ABB RobotStudio station: MGietka gripper.rspag

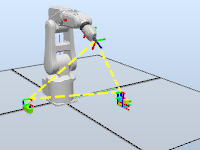
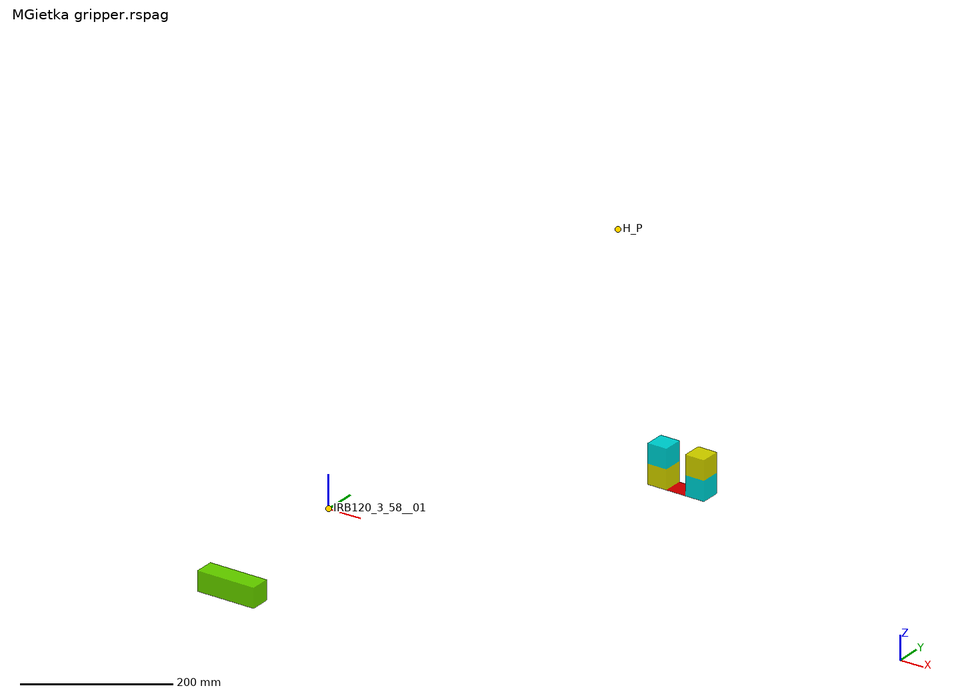
[picture v1: parts stored in the station drawn from their meshes, with robot base, taught points and paths (robot models come from the ABB library and are not in the file)]
--- station ---
Station PZPL zaliczenie 2 (saved by RobotStudio 21.4.9700.0)
Controller Controller1
  mechanical unit ROB_1: IRB120_3_58__01, 6 joints, base frame (0, 0, 0) mm
Layout (positions relative to the parent item):
  - IRB120_3_58__01 [mechanism, from Robots\IRB120_3_58_G_01.rslib] at (0, 0, 0) mm; joint values [0, 0, 0, 0, 0.5236, 0] (rad or m)
  - Smart_Gripper_Servo_Fingers [mechanism, from Tools\ABB_Smart_Gripper_Servo_Fingers.rslib] at (364.35, 0, 594) mm, rotated rx 180 ry 60 rz 180 deg; joint values [0.025] (rad or m)
  - Kosc_1 [part], size 30 x 30 x 30 mm
  - Kosc_2 [part], size 30 x 30 x 30 mm
  - Kosc_4 [part], size 30 x 30 x 30 mm
  - Kosc_3 [part], size 30 x 30 x 30 mm
  - podstawa [part], size 90 x 30 x 30 mm
  - PoseMover [smart component, from Components\PoseMover.rslib]
      properties: Mechanism=Smart_Gripper_Servo_Fingers; Pose=2; Duration=1
  - PoseMover_2 [smart component, from Components\PoseMover.rslib]
      properties: Mechanism=Smart_Gripper_Servo_Fingers; Pose=1; Duration=1
  - CollisionSensor [smart component, from Components\CollisionSensor.rslib]
      properties: Object1=Smart_Gripper_Servo_Fingers; Object2=Kosc_2; NearMiss=0; Part1=(none); Part2=(none); CollisionType=0
  - Attacher [smart component, from Components\Attacher.rslib]
      properties: Parent=Smart_Gripper_Servo_Fingers; Flange=0; Child=Kosc_2; Mount=false; Offset=[0 0 0]; Orientation=[0 0 0]
  - Detacher [smart component, from Components\Detacher.rslib]
      properties: Child=Kosc_2; KeepPosition=true
  - ClosestObject [smart component, from Components\ClosestObject.rslib]
      properties: ReferenceObject=Smart_Gripper_Servo_Fingers; ReferencePoint=[0 0 0]; RootObject=(none); ClosestObject=(none); ClosestPart=(none); Distance=0
  - plaszczyzna [part], size 90 x 30 x 0 mm
Attachment: Smart_Gripper_Servo_Fingers is attached to IRB120_3_58__01 / Link6
Attachment: Kosc1 is attached to Kosc_1
Attachment: Kosc_2 is attached to Kosc_2
Attachment: Kosc_3 is attached to Kosc_3
Attachment: Kosc_4 is attached to Kosc_4
Attachment: Podstawa is attached to podstawa
Attachment: Ramie is attached to IRB120_3_58__01 / Base
Station signals: DI start_s
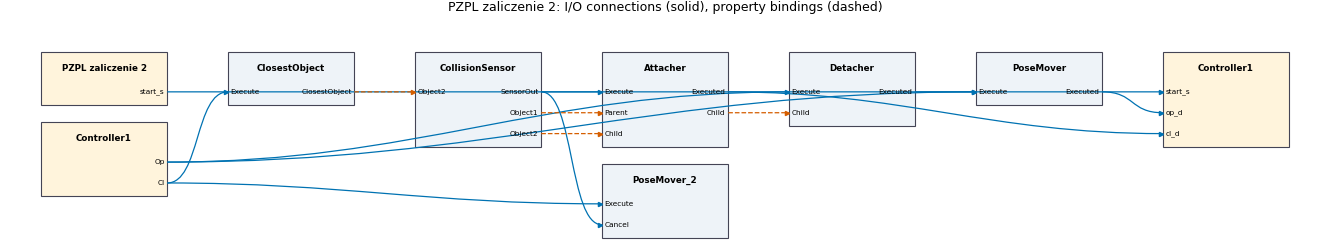
Station logic (signal -> signal, property => property):
  PZPL zaliczenie 2.start_s -> Controller1.start_s
  Controller1.Op -> PoseMover.Execute
  Controller1.Cl -> PoseMover_2.Execute
  CollisionSensor.SensorOut -> Attacher.Execute
  PoseMover.Executed -> Controller1.op_d
  CollisionSensor.SensorOut -> PoseMover_2.Cancel
  Controller1.Op -> Detacher.Execute
  Detacher.Executed -> PoseMover.Execute
  Attacher.Executed -> Controller1.cl_d
  Controller1.Cl -> ClosestObject.Execute
  CollisionSensor.Object1 => Attacher.Parent
  CollisionSensor.Object2 => Attacher.Child
  Attacher.Child => Detacher.Child
  ClosestObject.ClosestObject => CollisionSensor.Object2

--- Backups/Controller1/RAPID/TASK1/PROGMOD/CalibData.mod ---
MODULE CalibData
    PERS tooldata Servo:=[TRUE,[[0,0,114.2],[1,0,0,0]],[0.215,[8.7,12.3,49.2],[1,0,0,0],0.00021,0.00024,0.00009]];
    TASK PERS wobjdata Kosc1:=[FALSE,TRUE,"",[[300,300,0],[1,0,0,0]],[[0,0,0],[1,0,0,0]]];
    TASK PERS wobjdata Kosc_2:=[FALSE,TRUE,"",[[300,300,30],[1,0,0,0]],[[0,0,0],[1,0,0,0]]];
    TASK PERS wobjdata Kosc_3:=[FALSE,TRUE,"",[[360,300,0],[1,0,0,0]],[[0,0,0],[1,0,0,0]]];
    TASK PERS wobjdata Kosc_4:=[FALSE,TRUE,"",[[360,300,30],[1,0,0,0]],[[0,0,0],[1,0,0,0]]];
    TASK PERS wobjdata Podstawa:=[FALSE,TRUE,"",[[0,-300,0],[1,0,0,0]],[[0,0,0],[1,0,0,0]]];
    TASK PERS wobjdata Ramie:=[FALSE,TRUE,"",[[0,0,0],[1,0,0,0]],[[0,0,0],[1,0,0,0]]];
ENDMODULE

--- Backups/Controller1/RAPID/TASK1/PROGMOD/Module1.mod ---
MODULE Module1
    CONST robtarget H_P:=[[463.253930185,0,536.9],[0.5,0,0.866025404,0],[0,0,0,0],[9E+09,9E+09,9E+09,9E+09,9E+09,9E+09]];
    VAR robtarget Nad_kosc:=[[15,15,160],[0,1,0,0],[0,0,-2,0],[9E+09,9E+09,9E+09,9E+09,9E+09,9E+09]];
    VAR robtarget Kosc:=[[15,15,30],[0,1,0,0],[0,0,-2,0],[9E+09,9E+09,9E+09,9E+09,9E+09,9E+09]];
    VAR robtarget nad_cel:=[[75,15,160],[0,1,0,0],[-1,0,1,0],[9E+09,9E+09,9E+09,9E+09,9E+09,9E+09]];
    VAR robtarget cel:=[[75,15,60],[0,1,0,0],[-1,0,1,0],[9E+09,9E+09,9E+09,9E+09,9E+09,9E+09]];
    VAR num ilosc := 3;
!***********************************************************
    !
    ! Module:  Module1
    !
    ! Description:
    !   <Insert description here>
    !
    ! Author: Mati
    !
    ! Version: 1.0
    !
    !***********************************************************


    !***********************************************************
    !
    ! Procedure main
    !
    !   This is the entry point of your program
    !
    !***********************************************************
    PROC main()
        !Add your code here
    ENDPROC
    PROC Path_10()
            SetDO Cl,0;
            SetDO Op,0;
            WaitDI start_s,1;
            MoveJ H_P,v500,fine,Servo\WObj:=Ramie;
            MoveJ Nad_kosc,v500,fine,Servo\WObj:=Kosc_2;
            SetDO Op,1;
            WaitDI op_d,1;
            SetDO Op,0;
            MoveJ Kosc,v500,fine,Servo\WObj:=Kosc_2;
            SetDO Cl,1;
            WaitDI cl_d,1;
            SetDO Cl,0;
            MoveJ Nad_kosc,v500,fine,Servo\WObj:=Kosc_2;
            MoveJ nad_cel,v500,fine,Servo\WObj:=Podstawa;
            MoveJ cel,v500,fine,Servo\WObj:=Podstawa;
            SetDO Op,1;
            WaitDI op_d,1;
            SetDO Op,0;
            MoveJ nad_cel,v500,fine,Servo\WObj:=Podstawa;
            MoveJ H_P,v500,fine,Servo\WObj:=Ramie;
        FOR i FROM 1 TO ilosc DO
            IF (i MOD 2 = 0) THEN
                Kosc.trans.x := Kosc.trans.x - 60;
                Nad_kosc.trans.x := Nad_kosc.trans.x - 60;
                Kosc.trans.z := Kosc.trans.z - 30;

                cel.trans.x := cel.trans.x + 60;
                nad_cel.trans.x := nad_cel.trans.x + 60;
                cel.trans.z := cel.trans.z + 30;
            ELSE
                Kosc.trans.x := Kosc.trans.x + 60;
                Nad_kosc.trans.x := Nad_kosc.trans.x + 60;

                cel.trans.x := cel.trans.x - 60;
                nad_cel.trans.x := nad_cel.trans.x - 60;
            ENDIF
            SetDO Cl,0;
            SetDO Op,0;
            !WaitDI start_s,1;
            MoveJ H_P,v500,fine,Servo\WObj:=Ramie;
            MoveJ Nad_kosc,v500,fine,Servo\WObj:=Kosc_2;
            SetDO Op,1;
            WaitDI op_d,1;
            SetDO Op,0;
            MoveJ Kosc,v500,fine,Servo\WObj:=Kosc_2;
            SetDO Cl,1;
            WaitDI cl_d,1;
            SetDO Cl,0;
            MoveJ Nad_kosc,v500,fine,Servo\WObj:=Kosc_2;
            MoveJ nad_cel,v500,fine,Servo\WObj:=Podstawa;
            MoveJ cel,v500,fine,Servo\WObj:=Podstawa;
            SetDO Op,1;
            WaitDI op_d,1;
            SetDO Op,0;
            MoveJ nad_cel,v500,fine,Servo\WObj:=Podstawa;
            MoveJ H_P,v500,fine,Servo\WObj:=Ramie;
        ENDFOR
    ENDPROC
ENDMODULE

--- Backups/Controller1/SYSPAR/EIO.cfg ---
EIO:CFG_1.0:6:1::
#
EIO_SIGNAL:

      -Name "Op" -SignalType "DO"

      -Name "Cl" -SignalType "DO"

      -Name "op_d" -SignalType "DI"

      -Name "cl_d" -SignalType "DI"

      -Name "start_s" -SignalType "DI"
